// TIA Portal V17 export
// export: Created 2025-05-06T14:14:31.7335612Z, ExportSetting WithDefaults, DisplayName Totally Integrated Automation Portal, DisplayVersion V17 Update 8, DisplayName TIA Portal Openness, DisplayVersion V17 Update 8, DisplayName TIA Portal Version Control Interface, DisplayVersion V17, DisplayName SINAMICS Startdrive Advanced, DisplayVersion V17 SP2, DisplayName SINAMICS Startdrive G110M, G120, G120C, G120D, G120P, G115D, DisplayVersion V17 SP2, DisplayName SINAMICS Startdrive G130, G150, S120, S150, SINAMICS MV, S210, DisplayVersion V17 SP2, DisplayName STEP 7 Professional, DisplayVersion V17 Update 8, DisplayName SINUMERIK ONE STEP 7 Toolbox, DisplayVersion V17 Update 12, DisplayName SINUMERIK 840D sl STEP 7 Toolbox, DisplayVersion V17 Update 12, DisplayName STEP 7 Safety, DisplayVersion V17 Update 6, DisplayName WinCC Advanced, DisplayVersion V17 Update 8
FUNCTION_BLOCK "FB2003_CNC_MODES"   // FB2003, LAD
{ S7_Optimized_Access := 'TRUE' }
VERSION : 0.1
// stored: AutoNumber false, IsIECCheckEnabled false, IsRetainMemResEnabled false, MemoryReserve 100, SetENOAutomatically false, UDAEnableTagReadback false
   VAR_INPUT
      MODE_GROUP_NUMBER { ExternalAccessible := 'False'; ExternalVisible := 'False'; ExternalWritable := 'False'} : Int;   // MODE GROUP NUMBER
      MCH_RESET_FAULTS { ExternalAccessible := 'False'; ExternalVisible := 'False'; ExternalWritable := 'False'} : Bool;   // MACHINE RESET
      MDA_MODE_SLCTD { ExternalAccessible := 'False'; ExternalVisible := 'False'; ExternalWritable := 'False'} : Bool;   // MDA MODE SELECTED
      REF_MODE_SLCTD { ExternalAccessible := 'False'; ExternalVisible := 'False'; ExternalWritable := 'False'} : Bool;   // REFERENCE MODE SELECTED
      MODE_GROUP_GENERAL_DB { ExternalAccessible := 'False'; ExternalVisible := 'False'; ExternalWritable := 'False'} : "AUTO_SINGLE_SEMI_MANUAL";
   END_VAR
   VAR_OUTPUT
      ADDITIONAL_MODE_GROUP { ExternalAccessible := 'False'; ExternalVisible := 'False'; ExternalWritable := 'False'} : Struct
         A_AUTO { ExternalAccessible := 'False'; ExternalVisible := 'False'; ExternalWritable := 'False'} : Bool;
         A_MDA { ExternalAccessible := 'False'; ExternalVisible := 'False'; ExternalWritable := 'False'} : Bool;
         A_JOG { ExternalAccessible := 'False'; ExternalVisible := 'False'; ExternalWritable := 'False'} : Bool;
         f0_3 { ExternalAccessible := 'False'; ExternalVisible := 'False'; ExternalWritable := 'False'} : Bool;
         A_MCDisable { ExternalAccessible := 'False'; ExternalVisible := 'False'; ExternalWritable := 'False'} : Bool;
         A_MGStop { ExternalAccessible := 'False'; ExternalVisible := 'False'; ExternalWritable := 'False'} : Bool;
         A_MGStopASp { ExternalAccessible := 'False'; ExternalVisible := 'False'; ExternalWritable := 'False'} : Bool;
         A_MGReset { ExternalAccessible := 'False'; ExternalVisible := 'False'; ExternalWritable := 'False'} : Bool;
         A_TEACHIN { ExternalAccessible := 'False'; ExternalVisible := 'False'; ExternalWritable := 'False'} : Bool;
         A_REPOS { ExternalAccessible := 'False'; ExternalVisible := 'False'; ExternalWritable := 'False'} : Bool;
         A_REF { ExternalAccessible := 'False'; ExternalVisible := 'False'; ExternalWritable := 'False'} : Bool;
         f1_3 { ExternalAccessible := 'False'; ExternalVisible := 'False'; ExternalWritable := 'False'} : Bool;
         f1_4 { ExternalAccessible := 'False'; ExternalVisible := 'False'; ExternalWritable := 'False'} : Bool;
         f1_5 { ExternalAccessible := 'False'; ExternalVisible := 'False'; ExternalWritable := 'False'} : Bool;
         A_SingleBlock_B { ExternalAccessible := 'False'; ExternalVisible := 'False'; ExternalWritable := 'False'} : Bool;
         A_SingleBlock_A { ExternalAccessible := 'False'; ExternalVisible := 'False'; ExternalWritable := 'False'} : Bool;
         A_INC1 { ExternalAccessible := 'False'; ExternalVisible := 'False'; ExternalWritable := 'False'} : Bool;
         A_INC10 { ExternalAccessible := 'False'; ExternalVisible := 'False'; ExternalWritable := 'False'} : Bool;
         A_INC100 { ExternalAccessible := 'False'; ExternalVisible := 'False'; ExternalWritable := 'False'} : Bool;
         A_INC1000 { ExternalAccessible := 'False'; ExternalVisible := 'False'; ExternalWritable := 'False'} : Bool;
         A_INC10000 { ExternalAccessible := 'False'; ExternalVisible := 'False'; ExternalWritable := 'False'} : Bool;
         A_INCVar { ExternalAccessible := 'False'; ExternalVisible := 'False'; ExternalWritable := 'False'} : Bool;
         A_ContManTravel { ExternalAccessible := 'False'; ExternalVisible := 'False'; ExternalWritable := 'False'} : Bool;
         f2_7 { ExternalAccessible := 'False'; ExternalVisible := 'False'; ExternalWritable := 'False'} : Bool;
         f3 { ExternalAccessible := 'False'; ExternalVisible := 'False'; ExternalWritable := 'False'} : Byte;
         E_MMC_AUTO { ExternalAccessible := 'False'; ExternalVisible := 'False'; ExternalWritable := 'False'} : Bool;
         E_MMC_MDA { ExternalAccessible := 'False'; ExternalVisible := 'False'; ExternalWritable := 'False'} : Bool;
         E_MMC_JOG { ExternalAccessible := 'False'; ExternalVisible := 'False'; ExternalWritable := 'False'} : Bool;
         f4_3 { ExternalAccessible := 'False'; ExternalVisible := 'False'; ExternalWritable := 'False'} : Bool;
         f4_4 { ExternalAccessible := 'False'; ExternalVisible := 'False'; ExternalWritable := 'False'} : Bool;
         f4_5 { ExternalAccessible := 'False'; ExternalVisible := 'False'; ExternalWritable := 'False'} : Bool;
         f4_6 { ExternalAccessible := 'False'; ExternalVisible := 'False'; ExternalWritable := 'False'} : Bool;
         f4_7 { ExternalAccessible := 'False'; ExternalVisible := 'False'; ExternalWritable := 'False'} : Bool;
         E_MMC_TEACHIN { ExternalAccessible := 'False'; ExternalVisible := 'False'; ExternalWritable := 'False'} : Bool;
         E_MMC_REPOS { ExternalAccessible := 'False'; ExternalVisible := 'False'; ExternalWritable := 'False'} : Bool;
         E_MMC_REF { ExternalAccessible := 'False'; ExternalVisible := 'False'; ExternalWritable := 'False'} : Bool;
         f5_3 { ExternalAccessible := 'False'; ExternalVisible := 'False'; ExternalWritable := 'False'} : Bool;
         f5_4 { ExternalAccessible := 'False'; ExternalVisible := 'False'; ExternalWritable := 'False'} : Bool;
         f5_5 { ExternalAccessible := 'False'; ExternalVisible := 'False'; ExternalWritable := 'False'} : Bool;
         f5_6 { ExternalAccessible := 'False'; ExternalVisible := 'False'; ExternalWritable := 'False'} : Bool;
         f5_7 { ExternalAccessible := 'False'; ExternalVisible := 'False'; ExternalWritable := 'False'} : Bool;
         E_AUTO { ExternalAccessible := 'False'; ExternalVisible := 'False'; ExternalWritable := 'False'} : Bool;
         E_MDA { ExternalAccessible := 'False'; ExternalVisible := 'False'; ExternalWritable := 'False'} : Bool;
         E_JOG { ExternalAccessible := 'False'; ExternalVisible := 'False'; ExternalWritable := 'False'} : Bool;
         E_MGOK { ExternalAccessible := 'False'; ExternalVisible := 'False'; ExternalWritable := 'False'} : Bool;
         E_MGreseted { ExternalAccessible := 'False'; ExternalVisible := 'False'; ExternalWritable := 'False'} : Bool;
         E_NCKintJOG { ExternalAccessible := 'False'; ExternalVisible := 'False'; ExternalWritable := 'False'} : Bool;
         f6_6 { ExternalAccessible := 'False'; ExternalVisible := 'False'; ExternalWritable := 'False'} : Bool;
         E_ChanReset { ExternalAccessible := 'False'; ExternalVisible := 'False'; ExternalWritable := 'False'} : Bool;
         E_TEACHIN { ExternalAccessible := 'False'; ExternalVisible := 'False'; ExternalWritable := 'False'} : Bool;
         E_REPOS { ExternalAccessible := 'False'; ExternalVisible := 'False'; ExternalWritable := 'False'} : Bool;
         E_REF { ExternalAccessible := 'False'; ExternalVisible := 'False'; ExternalWritable := 'False'} : Bool;
         f7_3 { ExternalAccessible := 'False'; ExternalVisible := 'False'; ExternalWritable := 'False'} : Bool;
         f7_4 { ExternalAccessible := 'False'; ExternalVisible := 'False'; ExternalWritable := 'False'} : Bool;
         f7_5 { ExternalAccessible := 'False'; ExternalVisible := 'False'; ExternalWritable := 'False'} : Bool;
         f7_6 { ExternalAccessible := 'False'; ExternalVisible := 'False'; ExternalWritable := 'False'} : Bool;
         f7_7 { ExternalAccessible := 'False'; ExternalVisible := 'False'; ExternalWritable := 'False'} : Bool;
         E_INC1 { ExternalAccessible := 'False'; ExternalVisible := 'False'; ExternalWritable := 'False'} : Bool;
         E_INC10 { ExternalAccessible := 'False'; ExternalVisible := 'False'; ExternalWritable := 'False'} : Bool;
         E_INC100 { ExternalAccessible := 'False'; ExternalVisible := 'False'; ExternalWritable := 'False'} : Bool;
         E_INC1000 { ExternalAccessible := 'False'; ExternalVisible := 'False'; ExternalWritable := 'False'} : Bool;
         E_INC10000 { ExternalAccessible := 'False'; ExternalVisible := 'False'; ExternalWritable := 'False'} : Bool;
         E_INCVar { ExternalAccessible := 'False'; ExternalVisible := 'False'; ExternalWritable := 'False'} : Bool;
         E_ContManTravelAct { ExternalAccessible := 'False'; ExternalVisible := 'False'; ExternalWritable := 'False'} : Bool;
         f8_7 { ExternalAccessible := 'False'; ExternalVisible := 'False'; ExternalWritable := 'False'} : Bool;
         f9 { ExternalAccessible := 'False'; ExternalVisible := 'False'; ExternalWritable := 'False'} : Byte;
         E_HMI_INC1 { ExternalAccessible := 'False'; ExternalVisible := 'False'; ExternalWritable := 'False'} : Bool;
         E_HMI_INC10 { ExternalAccessible := 'False'; ExternalVisible := 'False'; ExternalWritable := 'False'} : Bool;
         E_HMI_INC100 { ExternalAccessible := 'False'; ExternalVisible := 'False'; ExternalWritable := 'False'} : Bool;
         E_HMI_INC1000 { ExternalAccessible := 'False'; ExternalVisible := 'False'; ExternalWritable := 'False'} : Bool;
         E_HMI_INC10000 { ExternalAccessible := 'False'; ExternalVisible := 'False'; ExternalWritable := 'False'} : Bool;
         E_HMI_INCVar { ExternalAccessible := 'False'; ExternalVisible := 'False'; ExternalWritable := 'False'} : Bool;
         E_HMI_ContManTravel { ExternalAccessible := 'False'; ExternalVisible := 'False'; ExternalWritable := 'False'} : Bool;
         f10_7 { ExternalAccessible := 'False'; ExternalVisible := 'False'; ExternalWritable := 'False'} : Bool;
         f11 { ExternalAccessible := 'False'; ExternalVisible := 'False'; ExternalWritable := 'False'} : Byte;
         f12 { ExternalAccessible := 'False'; ExternalVisible := 'False'; ExternalWritable := 'False'} : Array[12..19] of Byte;
      END_STRUCT;
   END_VAR
   VAR_TEMP   // added for the SCL form of the ladder/FBD networks
      _w1 : Bool;
   END_VAR
BEGIN

NETWORK
TITLE = ACTUAL VALUE IN WCS 0=MCS / Actual value in WCS 0=MCS
// WKS/MKS

      AN    "LBP_HMI".E_ActWCS;
      JC    M001;
      AN    "LBP_HMI".A_ActWCS;
      =     "LBP_HMI".A_ActWCS;
      CLR;
      =     "LBP_HMI".E_ActWCS;
M001: NOP   0;

REGION Network 2: MODE GROUP RESET / Mode group reset
   // BAG Reset
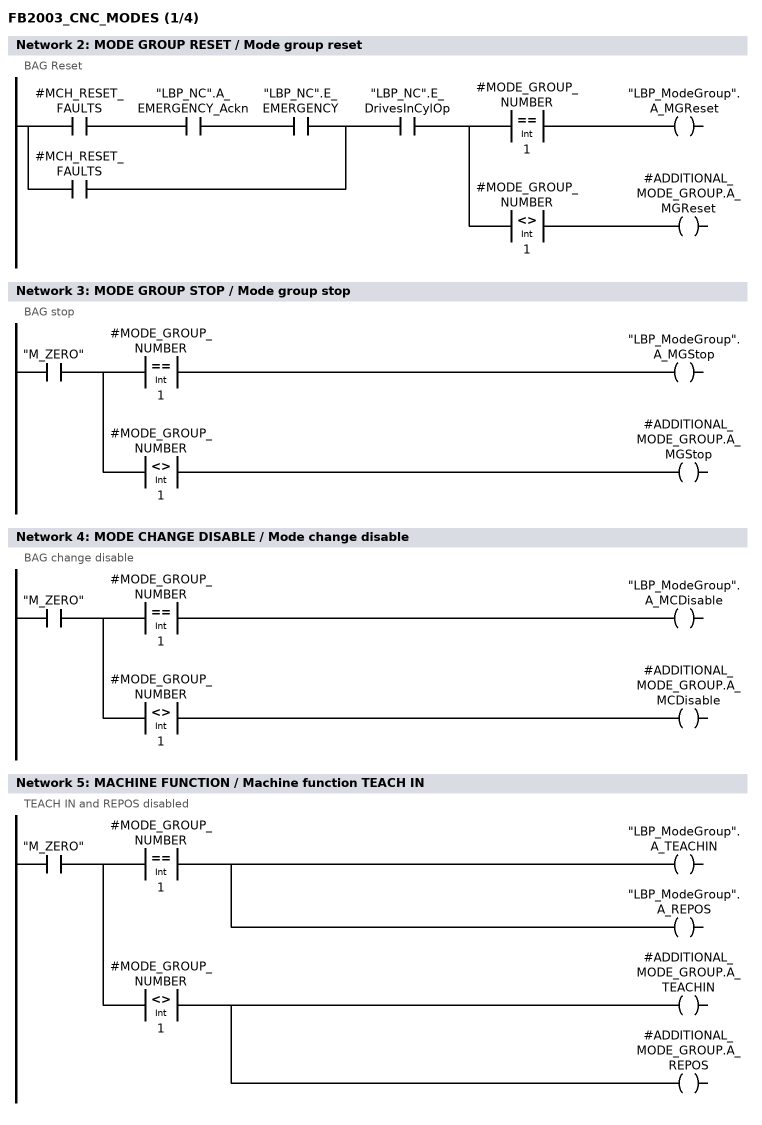
   RUNG wire#powerrail
      Contact( #MCH_RESET_FAULTS )
      Contact( "LBP_NC".A_EMERGENCY_Ackn )
      Contact( "LBP_NC".E_EMERGENCY )
      wire#w1
      Contact( "LBP_NC".E_DrivesInCylOp )
      wire#w2
      { S7_Templates := "SrcType := Int" } EQ_Contact(in1 := #MODE_GROUP_NUMBER, in2 := 1)
      Coil( "LBP_ModeGroup".A_MGReset )
   END_RUNG
   RUNG wire#powerrail
      Contact( #MCH_RESET_FAULTS )
   END_RUNG wire#w1
   RUNG wire#w2
      { S7_Templates := "SrcType := Int" } NE_Contact(in1 := #MODE_GROUP_NUMBER, in2 := 1)
      Coil( #ADDITIONAL_MODE_GROUP.A_MGReset )
   END_RUNG
   // the same network as SCL:
   #_w1 := ((#MCH_RESET_FAULTS AND "LBP_NC".A_EMERGENCY_Ackn AND "LBP_NC".E_EMERGENCY) OR #MCH_RESET_FAULTS) AND "LBP_NC".E_DrivesInCylOp;
   "LBP_ModeGroup".A_MGReset := #_w1 AND (#MODE_GROUP_NUMBER = 1);
   #ADDITIONAL_MODE_GROUP.A_MGReset := #_w1 AND (#MODE_GROUP_NUMBER <> 1);
END_REGION

REGION Network 3: MODE GROUP STOP / Mode group stop
   // BAG stop
   RUNG wire#powerrail
      Contact( "M_ZERO" )
      wire#w1
      { S7_Templates := "SrcType := Int" } EQ_Contact(in1 := #MODE_GROUP_NUMBER, in2 := 1)
      Coil( "LBP_ModeGroup".A_MGStop )
   END_RUNG
   RUNG wire#w1
      { S7_Templates := "SrcType := Int" } NE_Contact(in1 := #MODE_GROUP_NUMBER, in2 := 1)
      Coil( #ADDITIONAL_MODE_GROUP.A_MGStop )
   END_RUNG
   // the same network as SCL:
   "LBP_ModeGroup".A_MGStop := "M_ZERO" AND (#MODE_GROUP_NUMBER = 1);
   #ADDITIONAL_MODE_GROUP.A_MGStop := "M_ZERO" AND (#MODE_GROUP_NUMBER <> 1);
END_REGION

REGION Network 4: MODE CHANGE DISABLE / Mode change disable
   // BAG change disable
   RUNG wire#powerrail
      Contact( "M_ZERO" )
      wire#w1
      { S7_Templates := "SrcType := Int" } EQ_Contact(in1 := #MODE_GROUP_NUMBER, in2 := 1)
      Coil( "LBP_ModeGroup".A_MCDisable )
   END_RUNG
   RUNG wire#w1
      { S7_Templates := "SrcType := Int" } NE_Contact(in1 := #MODE_GROUP_NUMBER, in2 := 1)
      Coil( #ADDITIONAL_MODE_GROUP.A_MCDisable )
   END_RUNG
   // the same network as SCL:
   "LBP_ModeGroup".A_MCDisable := "M_ZERO" AND (#MODE_GROUP_NUMBER = 1);
   #ADDITIONAL_MODE_GROUP.A_MCDisable := "M_ZERO" AND (#MODE_GROUP_NUMBER <> 1);
END_REGION

REGION Network 5: MACHINE FUNCTION / Machine function TEACH IN
   // TEACH IN and REPOS disabled
   RUNG wire#powerrail
      Contact( "M_ZERO" )
      wire#w1
      { S7_Templates := "SrcType := Int" } EQ_Contact(in1 := #MODE_GROUP_NUMBER, in2 := 1)
      wire#w2
      Coil( "LBP_ModeGroup".A_TEACHIN )
   END_RUNG
   RUNG wire#w2
      Coil( "LBP_ModeGroup".A_REPOS )
   END_RUNG
   RUNG wire#w1
      { S7_Templates := "SrcType := Int" } NE_Contact(in1 := #MODE_GROUP_NUMBER, in2 := 1)
      wire#w3
      Coil( #ADDITIONAL_MODE_GROUP.A_TEACHIN )
   END_RUNG
   RUNG wire#w3
      Coil( #ADDITIONAL_MODE_GROUP.A_REPOS )
   END_RUNG
   // the same network as SCL:
   "LBP_ModeGroup".A_TEACHIN := "M_ZERO" AND (#MODE_GROUP_NUMBER = 1);
   "LBP_ModeGroup".A_REPOS := "LBP_ModeGroup".A_TEACHIN;
   #ADDITIONAL_MODE_GROUP.A_TEACHIN := "M_ZERO" AND (#MODE_GROUP_NUMBER <> 1);
   #ADDITIONAL_MODE_GROUP.A_REPOS := #ADDITIONAL_MODE_GROUP.A_TEACHIN;
END_REGION

REGION Network 6: OPERATING MODE AUTOMATIC / AUTOMATIC MODE
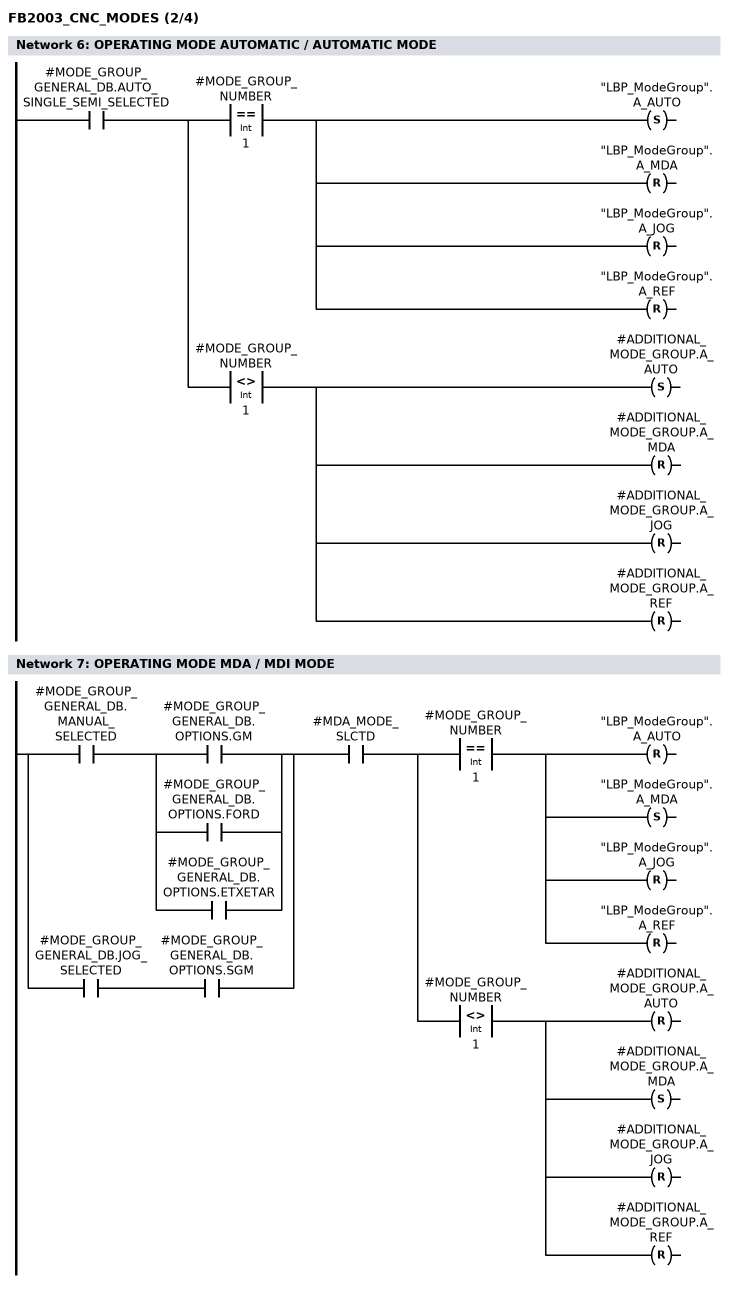
   RUNG wire#powerrail
      Contact( #MODE_GROUP_GENERAL_DB.AUTO_SINGLE_SEMI_SELECTED )
      wire#w1
      { S7_Templates := "SrcType := Int" } EQ_Contact(in1 := #MODE_GROUP_NUMBER, in2 := 1)
      wire#w2
      S_Coil( "LBP_ModeGroup".A_AUTO )
   END_RUNG
   RUNG wire#w2
      R_Coil( "LBP_ModeGroup".A_MDA )
   END_RUNG
   RUNG wire#w2
      R_Coil( "LBP_ModeGroup".A_JOG )
   END_RUNG
   RUNG wire#w2
      R_Coil( "LBP_ModeGroup".A_REF )
   END_RUNG
   RUNG wire#w1
      { S7_Templates := "SrcType := Int" } NE_Contact(in1 := #MODE_GROUP_NUMBER, in2 := 1)
      wire#w3
      S_Coil( #ADDITIONAL_MODE_GROUP.A_AUTO )
   END_RUNG
   RUNG wire#w3
      R_Coil( #ADDITIONAL_MODE_GROUP.A_MDA )
   END_RUNG
   RUNG wire#w3
      R_Coil( #ADDITIONAL_MODE_GROUP.A_JOG )
   END_RUNG
   RUNG wire#w3
      R_Coil( #ADDITIONAL_MODE_GROUP.A_REF )
   END_RUNG
   // the same network as SCL:
   IF #MODE_GROUP_GENERAL_DB.AUTO_SINGLE_SEMI_SELECTED AND (#MODE_GROUP_NUMBER = 1) THEN
       "LBP_ModeGroup".A_AUTO := TRUE;
       "LBP_ModeGroup".A_MDA := FALSE;
       "LBP_ModeGroup".A_JOG := FALSE;
       "LBP_ModeGroup".A_REF := FALSE;
   END_IF;
   IF #MODE_GROUP_GENERAL_DB.AUTO_SINGLE_SEMI_SELECTED AND (#MODE_GROUP_NUMBER <> 1) THEN
       #ADDITIONAL_MODE_GROUP.A_AUTO := TRUE;
       #ADDITIONAL_MODE_GROUP.A_MDA := FALSE;
       #ADDITIONAL_MODE_GROUP.A_JOG := FALSE;
       #ADDITIONAL_MODE_GROUP.A_REF := FALSE;
   END_IF;
END_REGION

REGION Network 7: OPERATING MODE MDA / MDI MODE
   RUNG wire#powerrail
      Contact( #MODE_GROUP_GENERAL_DB.MANUAL_SELECTED )
      wire#w1
      Contact( #MODE_GROUP_GENERAL_DB.OPTIONS.GM )
      wire#w2
      Contact( #MDA_MODE_SLCTD )
      wire#w3
      { S7_Templates := "SrcType := Int" } EQ_Contact(in1 := #MODE_GROUP_NUMBER, in2 := 1)
      wire#w4
      R_Coil( "LBP_ModeGroup".A_AUTO )
   END_RUNG
   RUNG wire#w1
      Contact( #MODE_GROUP_GENERAL_DB.OPTIONS.FORD )
   END_RUNG wire#w2
   RUNG wire#w1
      Contact( #MODE_GROUP_GENERAL_DB.OPTIONS.ETXETAR )
   END_RUNG wire#w2
   RUNG wire#powerrail
      Contact( #MODE_GROUP_GENERAL_DB.JOG_SELECTED )
      Contact( #MODE_GROUP_GENERAL_DB.OPTIONS.SGM )
   END_RUNG wire#w2
   RUNG wire#w4
      S_Coil( "LBP_ModeGroup".A_MDA )
   END_RUNG
   RUNG wire#w4
      R_Coil( "LBP_ModeGroup".A_JOG )
   END_RUNG
   RUNG wire#w4
      R_Coil( "LBP_ModeGroup".A_REF )
   END_RUNG
   RUNG wire#w3
      { S7_Templates := "SrcType := Int" } NE_Contact(in1 := #MODE_GROUP_NUMBER, in2 := 1)
      wire#w5
      R_Coil( #ADDITIONAL_MODE_GROUP.A_AUTO )
   END_RUNG
   RUNG wire#w5
      S_Coil( #ADDITIONAL_MODE_GROUP.A_MDA )
   END_RUNG
   RUNG wire#w5
      R_Coil( #ADDITIONAL_MODE_GROUP.A_JOG )
   END_RUNG
   RUNG wire#w5
      R_Coil( #ADDITIONAL_MODE_GROUP.A_REF )
   END_RUNG
   // the same network as SCL:
   #_w1 := ((#MODE_GROUP_GENERAL_DB.MANUAL_SELECTED AND (#MODE_GROUP_GENERAL_DB.OPTIONS.GM OR #MODE_GROUP_GENERAL_DB.OPTIONS.FORD OR #MODE_GROUP_GENERAL_DB.OPTIONS.ETXETAR)) OR (#MODE_GROUP_GENERAL_DB.JOG_SELECTED AND #MODE_GROUP_GENERAL_DB.OPTIONS.SGM)) AND #MDA_MODE_SLCTD;
   IF #_w1 AND (#MODE_GROUP_NUMBER = 1) THEN
       "LBP_ModeGroup".A_AUTO := FALSE;
       "LBP_ModeGroup".A_MDA := TRUE;
       "LBP_ModeGroup".A_JOG := FALSE;
       "LBP_ModeGroup".A_REF := FALSE;
   END_IF;
   IF #_w1 AND (#MODE_GROUP_NUMBER <> 1) THEN
       #ADDITIONAL_MODE_GROUP.A_AUTO := FALSE;
       #ADDITIONAL_MODE_GROUP.A_MDA := TRUE;
       #ADDITIONAL_MODE_GROUP.A_JOG := FALSE;
       #ADDITIONAL_MODE_GROUP.A_REF := FALSE;
   END_IF;
END_REGION

REGION Network 8: OPERATING MODE MANUAL / JOG MODE
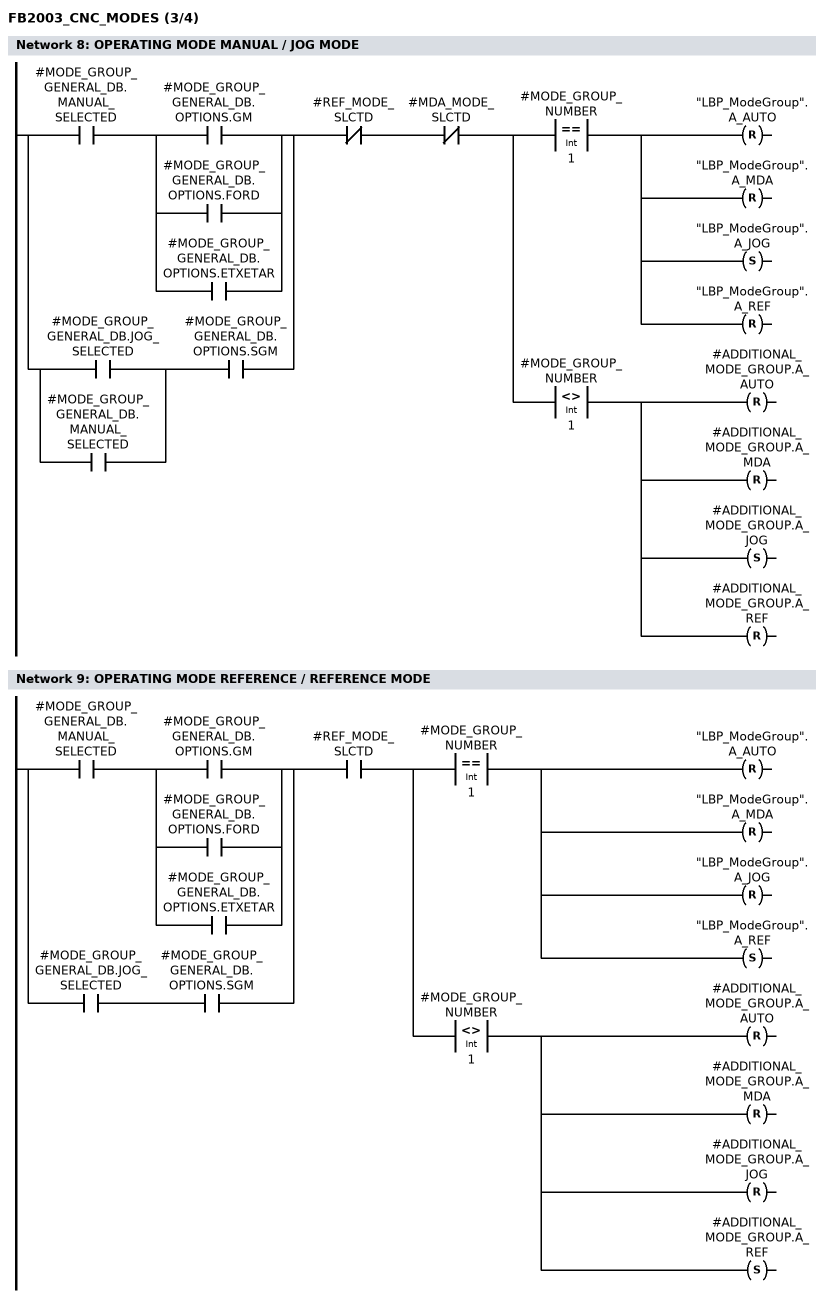
   RUNG wire#powerrail
      Contact( #MODE_GROUP_GENERAL_DB.MANUAL_SELECTED )
      wire#w1
      Contact( #MODE_GROUP_GENERAL_DB.OPTIONS.GM )
      wire#w2
      I_Contact( #REF_MODE_SLCTD )
      I_Contact( #MDA_MODE_SLCTD )
      wire#w4
      { S7_Templates := "SrcType := Int" } EQ_Contact(in1 := #MODE_GROUP_NUMBER, in2 := 1)
      wire#w5
      R_Coil( "LBP_ModeGroup".A_AUTO )
   END_RUNG
   RUNG wire#w1
      Contact( #MODE_GROUP_GENERAL_DB.OPTIONS.FORD )
   END_RUNG wire#w2
   RUNG wire#w1
      Contact( #MODE_GROUP_GENERAL_DB.OPTIONS.ETXETAR )
   END_RUNG wire#w2
   RUNG wire#powerrail
      Contact( #MODE_GROUP_GENERAL_DB.JOG_SELECTED )
      wire#w3
      Contact( #MODE_GROUP_GENERAL_DB.OPTIONS.SGM )
   END_RUNG wire#w2
   RUNG wire#powerrail
      Contact( #MODE_GROUP_GENERAL_DB.MANUAL_SELECTED )
   END_RUNG wire#w3
   RUNG wire#w5
      R_Coil( "LBP_ModeGroup".A_MDA )
   END_RUNG
   RUNG wire#w5
      S_Coil( "LBP_ModeGroup".A_JOG )
   END_RUNG
   RUNG wire#w5
      R_Coil( "LBP_ModeGroup".A_REF )
   END_RUNG
   RUNG wire#w4
      { S7_Templates := "SrcType := Int" } NE_Contact(in1 := #MODE_GROUP_NUMBER, in2 := 1)
      wire#w6
      R_Coil( #ADDITIONAL_MODE_GROUP.A_AUTO )
   END_RUNG
   RUNG wire#w6
      R_Coil( #ADDITIONAL_MODE_GROUP.A_MDA )
   END_RUNG
   RUNG wire#w6
      S_Coil( #ADDITIONAL_MODE_GROUP.A_JOG )
   END_RUNG
   RUNG wire#w6
      R_Coil( #ADDITIONAL_MODE_GROUP.A_REF )
   END_RUNG
   // the same network as SCL:
   #_w1 := ((#MODE_GROUP_GENERAL_DB.MANUAL_SELECTED AND (#MODE_GROUP_GENERAL_DB.OPTIONS.GM OR #MODE_GROUP_GENERAL_DB.OPTIONS.FORD OR #MODE_GROUP_GENERAL_DB.OPTIONS.ETXETAR)) OR ((#MODE_GROUP_GENERAL_DB.JOG_SELECTED OR #MODE_GROUP_GENERAL_DB.MANUAL_SELECTED) AND #MODE_GROUP_GENERAL_DB.OPTIONS.SGM)) AND NOT #REF_MODE_SLCTD AND NOT #MDA_MODE_SLCTD;
   IF #_w1 AND (#MODE_GROUP_NUMBER = 1) THEN
       "LBP_ModeGroup".A_AUTO := FALSE;
       "LBP_ModeGroup".A_MDA := FALSE;
       "LBP_ModeGroup".A_JOG := TRUE;
       "LBP_ModeGroup".A_REF := FALSE;
   END_IF;
   IF #_w1 AND (#MODE_GROUP_NUMBER <> 1) THEN
       #ADDITIONAL_MODE_GROUP.A_AUTO := FALSE;
       #ADDITIONAL_MODE_GROUP.A_MDA := FALSE;
       #ADDITIONAL_MODE_GROUP.A_JOG := TRUE;
       #ADDITIONAL_MODE_GROUP.A_REF := FALSE;
   END_IF;
END_REGION

REGION Network 9: OPERATING MODE REFERENCE / REFERENCE MODE
   RUNG wire#powerrail
      Contact( #MODE_GROUP_GENERAL_DB.MANUAL_SELECTED )
      wire#w1
      Contact( #MODE_GROUP_GENERAL_DB.OPTIONS.GM )
      wire#w2
      Contact( #REF_MODE_SLCTD )
      wire#w3
      { S7_Templates := "SrcType := Int" } EQ_Contact(in1 := #MODE_GROUP_NUMBER, in2 := 1)
      wire#w4
      R_Coil( "LBP_ModeGroup".A_AUTO )
   END_RUNG
   RUNG wire#w1
      Contact( #MODE_GROUP_GENERAL_DB.OPTIONS.FORD )
   END_RUNG wire#w2
   RUNG wire#w1
      Contact( #MODE_GROUP_GENERAL_DB.OPTIONS.ETXETAR )
   END_RUNG wire#w2
   RUNG wire#powerrail
      Contact( #MODE_GROUP_GENERAL_DB.JOG_SELECTED )
      Contact( #MODE_GROUP_GENERAL_DB.OPTIONS.SGM )
   END_RUNG wire#w2
   RUNG wire#w4
      R_Coil( "LBP_ModeGroup".A_MDA )
   END_RUNG
   RUNG wire#w4
      R_Coil( "LBP_ModeGroup".A_JOG )
   END_RUNG
   RUNG wire#w4
      S_Coil( "LBP_ModeGroup".A_REF )
   END_RUNG
   RUNG wire#w3
      { S7_Templates := "SrcType := Int" } NE_Contact(in1 := #MODE_GROUP_NUMBER, in2 := 1)
      wire#w5
      R_Coil( #ADDITIONAL_MODE_GROUP.A_AUTO )
   END_RUNG
   RUNG wire#w5
      R_Coil( #ADDITIONAL_MODE_GROUP.A_MDA )
   END_RUNG
   RUNG wire#w5
      R_Coil( #ADDITIONAL_MODE_GROUP.A_JOG )
   END_RUNG
   RUNG wire#w5
      S_Coil( #ADDITIONAL_MODE_GROUP.A_REF )
   END_RUNG
   // the same network as SCL:
   #_w1 := ((#MODE_GROUP_GENERAL_DB.MANUAL_SELECTED AND (#MODE_GROUP_GENERAL_DB.OPTIONS.GM OR #MODE_GROUP_GENERAL_DB.OPTIONS.FORD OR #MODE_GROUP_GENERAL_DB.OPTIONS.ETXETAR)) OR (#MODE_GROUP_GENERAL_DB.JOG_SELECTED AND #MODE_GROUP_GENERAL_DB.OPTIONS.SGM)) AND #REF_MODE_SLCTD;
   IF #_w1 AND (#MODE_GROUP_NUMBER = 1) THEN
       "LBP_ModeGroup".A_AUTO := FALSE;
       "LBP_ModeGroup".A_MDA := FALSE;
       "LBP_ModeGroup".A_JOG := FALSE;
       "LBP_ModeGroup".A_REF := TRUE;
   END_IF;
   IF #_w1 AND (#MODE_GROUP_NUMBER <> 1) THEN
       #ADDITIONAL_MODE_GROUP.A_AUTO := FALSE;
       #ADDITIONAL_MODE_GROUP.A_MDA := FALSE;
       #ADDITIONAL_MODE_GROUP.A_JOG := FALSE;
       #ADDITIONAL_MODE_GROUP.A_REF := TRUE;
   END_IF;
END_REGION

REGION Network 10: OPERATING MODE NO MODE / NO REFERENCE MODE
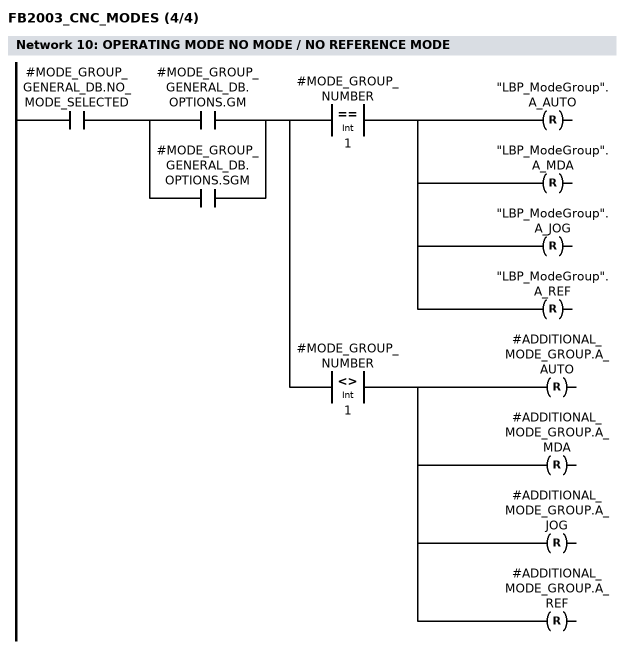
   RUNG wire#powerrail
      Contact( #MODE_GROUP_GENERAL_DB.NO_MODE_SELECTED )
      wire#w1
      Contact( #MODE_GROUP_GENERAL_DB.OPTIONS.GM )
      wire#w2
      { S7_Templates := "SrcType := Int" } EQ_Contact(in1 := #MODE_GROUP_NUMBER, in2 := 1)
      wire#w3
      R_Coil( "LBP_ModeGroup".A_AUTO )
   END_RUNG
   RUNG wire#w1
      Contact( #MODE_GROUP_GENERAL_DB.OPTIONS.SGM )
   END_RUNG wire#w2
   RUNG wire#w3
      R_Coil( "LBP_ModeGroup".A_MDA )
   END_RUNG
   RUNG wire#w3
      R_Coil( "LBP_ModeGroup".A_JOG )
   END_RUNG
   RUNG wire#w3
      R_Coil( "LBP_ModeGroup".A_REF )
   END_RUNG
   RUNG wire#w2
      { S7_Templates := "SrcType := Int" } NE_Contact(in1 := #MODE_GROUP_NUMBER, in2 := 1)
      wire#w4
      R_Coil( #ADDITIONAL_MODE_GROUP.A_AUTO )
   END_RUNG
   RUNG wire#w4
      R_Coil( #ADDITIONAL_MODE_GROUP.A_MDA )
   END_RUNG
   RUNG wire#w4
      R_Coil( #ADDITIONAL_MODE_GROUP.A_JOG )
   END_RUNG
   RUNG wire#w4
      R_Coil( #ADDITIONAL_MODE_GROUP.A_REF )
   END_RUNG
   // the same network as SCL:
   #_w1 := #MODE_GROUP_GENERAL_DB.NO_MODE_SELECTED AND (#MODE_GROUP_GENERAL_DB.OPTIONS.GM OR #MODE_GROUP_GENERAL_DB.OPTIONS.SGM);
   IF #_w1 AND (#MODE_GROUP_NUMBER = 1) THEN
       "LBP_ModeGroup".A_AUTO := FALSE;
       "LBP_ModeGroup".A_MDA := FALSE;
       "LBP_ModeGroup".A_JOG := FALSE;
       "LBP_ModeGroup".A_REF := FALSE;
   END_IF;
   IF #_w1 AND (#MODE_GROUP_NUMBER <> 1) THEN
       #ADDITIONAL_MODE_GROUP.A_AUTO := FALSE;
       #ADDITIONAL_MODE_GROUP.A_MDA := FALSE;
       #ADDITIONAL_MODE_GROUP.A_JOG := FALSE;
       #ADDITIONAL_MODE_GROUP.A_REF := FALSE;
   END_IF;
END_REGION
END_FUNCTION_BLOCK
